PROGRAM MAIN
VAR
	input :BOOL;
	output : BOOL;
	
END_VAR

Lamp ();
Light();

END_PROGRAM

(* stored: Version 1.1.0.1, ProductVersion 3.1.4024.12
   POU MAIN: Id {2babdd2d-5622-4c41-b52e-13838c2e5e51}, SpecialFunc None *)
